// TIA Portal V18 export
FUNCTION "Sunc_2" : Void   // FC4, LAD
{ S7_Optimized_Access := 'TRUE' }
VERSION : 0.1
// stored: AutoNumber true, IsIECCheckEnabled false, SetENOAutomatically false, UDAEnableTagReadback false
BEGIN

REGION Network 1
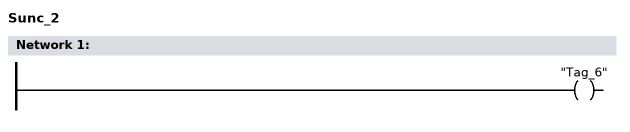
   RUNG wire#powerrail
      Coil( "Tag_6" )
   END_RUNG
   // the same network as SCL:
   "Tag_6" := TRUE;
END_REGION
END_FUNCTION
